// TIA Portal V20 program export: 1 tag tables, 0 data types, 1 data blocks, 6 code blocks (in call order from the OBs), 0 instance data blocks

VAR_GLOBAL   // PLC tag table "Default tag table"
   System_Byte AT %MB1 : Byte;
   FirstScan AT %M1.0 : Bool;
   DiagStatusUpdate AT %M1.1 : Bool;
   AlwaysTRUE AT %M1.2 : Bool;
   AlwaysFALSE AT %M1.3 : Bool;
   Clock_Byte AT %MB0 : Byte;
   Clock_10Hz AT %M0.0 : Bool;
   Clock_5Hz AT %M0.1 : Bool;
   "Clock_2.5Hz" AT %M0.2 : Bool;
   Clock_2Hz AT %M0.3 : Bool;
   "Clock_1.25Hz" AT %M0.4 : Bool;
   Clock_1Hz AT %M0.5 : Bool;
   "Clock_0.625Hz" AT %M0.6 : Bool;
   "Clock_0.5Hz" AT %M0.7 : Bool;
   AAA AT %M2.0 : Bool;
END_VAR

DATA_BLOCK "Data_block_1"   // DB1
{ S7_Optimized_Access := 'TRUE' }
// stored: MemoryReserve 100
   VAR
      "A" : Bool;
      "B" : Bool;
      C : Bool;
   END_VAR
BEGIN
END_DATA_BLOCK

ORGANIZATION_BLOCK "Main"   // OB1, LAD, ProgramCycle
TITLE = "Main Program Sweep (Cycle)"
{ S7_Optimized_Access := 'TRUE' }
// stored: SetENOAutomatically false
   VAR_INPUT
      Initial_Call : Bool;   // Initial call of this OB
      Remanence : Bool;   // =True, if remanent data are available
   END_VAR
   VAR_TEMP   // added for the SCL form of the ladder/FBD networks
      _w1 : Bool;
   END_VAR
BEGIN

REGION Network 1
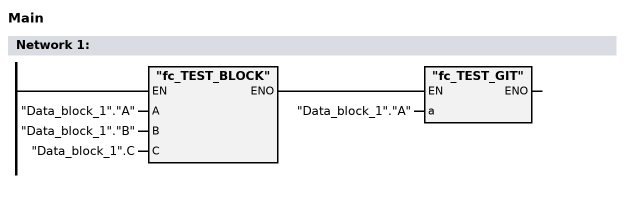
   RUNG wire#powerrail
      "fc_TEST_BLOCK"("A" := "Data_block_1"."A", "B" := "Data_block_1"."B", C := "Data_block_1".C)
      "fc_TEST_GIT"("a" := "Data_block_1"."A")
   END_RUNG
   // the same network as SCL:
   "fc_TEST_BLOCK"("A" := "Data_block_1"."A", "B" := "Data_block_1"."B", C := "Data_block_1".C, ENO => #_w1);
   IF #_w1 THEN "fc_TEST_GIT"("a" := "Data_block_1"."A"); END_IF;
END_REGION
END_ORGANIZATION_BLOCK

FUNCTION "fc_TEST_BLOCK" : Void
TITLE = MOJ_BLOCK_TESTOWY
{ S7_Optimized_Access := 'TRUE' }
AUTHOR : PJO
FAMILY : BLOKI_TESTOWE
VERSION : 0.1
//ZOBACZYMY TEGO EFEKT
   VAR_INPUT 
      A : Bool;
      B : Bool;
      C : Bool;
   END_VAR


BEGIN
	REGION BLOCK_TESTOWY
	    IF #A THEN
	        #B := TRUE;
	    // ELSE
	    //     #B := FALSE;
	    //     /dodalem komentarz
	    END_IF;
	END_REGION
	
END_FUNCTION

FUNCTION "fc_TEST_GIT" : Void
{ S7_Optimized_Access := 'TRUE' }
VERSION : 0.1
   VAR_IN_OUT 
      a : Bool;
   END_VAR


BEGIN
	IF #a THEN
	    #a := NOT #a;
	END_IF;
	
END_FUNCTION

FUNCTION "fc" : Bool
{ S7_Optimized_Access := 'TRUE' }
VERSION : 0.1
   VAR_INPUT 
      a : Bool;
   END_VAR


BEGIN
	#fc := NOT #a;
END_FUNCTION

FUNCTION "fc_BRANCH_A" : Void
{ S7_Optimized_Access := 'TRUE' }
VERSION : 0.1

BEGIN
END_FUNCTION

FUNCTION "fc_BRANCH_B" : Void
{ S7_Optimized_Access := 'TRUE' }
VERSION : 0.1

BEGIN
END_FUNCTION
